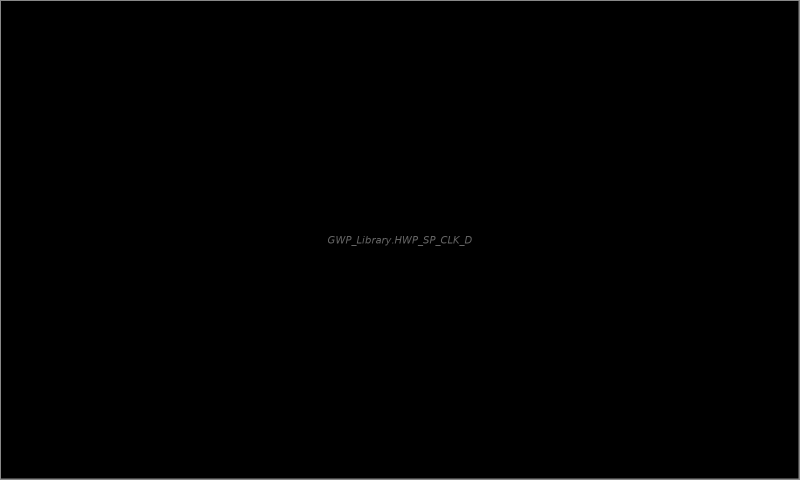
VISUALIZATION HWP_SP_CLK_D  // 800x480
    Frame (0,0 800x480)
        shows GWP_Library.HWP_SP_CLK_D(FB_CLK_D := Main.HWP_SP_0.GR_4_ohne_RE_0.TagNacht, FB_Init_1 := Main.Init_0)
END_VISUALIZATION

(* stored: Version 1.1.0.1, ProductVersion 3.1.4022.6
   Visu HWP_SP_CLK_D: Id {ea4260a6-fa79-4406-849f-334e0a7fc5ad} *)
